// Block: WeldReg_PERS

DATA_BLOCK WeldReg_PERS
VERSION : 0.1
   NON_RETAIN
   VAR
      PersistentValues : udt_WeldReg_Pers;
   END_VAR

BEGIN
   // No initialization required
END_DATA_BLOCK
